Fanuc KAREL source: kc00026.KL

-- PROVISIONAL review KL for V940-1; original PC SHA256 9882130c3fa4ab0798106e8d5d1c845b52d76eb7248f879cbfec3ecfef4f3993
-- Incomplete behavior may be omitted. Consult companion uncertainty JSON. Do not deploy.
PROGRAM KC00026
%NOLOCKGROUP
BEGIN
  -- V9_ZERO_TABLE_METADATA_HINT layout=0002_ascii; no indexed target words; source/name/runtime held
  -- UNRESOLVED_PC offsets 5-45; opcodes 27,22,22,22,22,22,22,31
  -- UNRESOLVED_PC offsets 50-54; opcodes 7F
END KC00026
